// TIA Portal V17 export
// export: Created 2025-05-22T05:59:44.8642244Z, ExportSetting WithDefaults, DisplayName Totally Integrated Automation Portal, DisplayVersion V17 Update 8, DisplayName TIA Portal Openness, DisplayVersion V17 Update 8, DisplayName TIA Portal Version Control Interface, DisplayVersion V17, DisplayName SINAMICS Startdrive Advanced, DisplayVersion V17 SP2, DisplayName SINAMICS Startdrive G110M, G120, G120C, G120D, G120P, G115D, DisplayVersion V17 SP2, DisplayName SINAMICS Startdrive G130, G150, S120, S150, SINAMICS MV, S210, DisplayVersion V17 SP2, DisplayName STEP 7 Professional, DisplayVersion V17 Update 8, DisplayName SINUMERIK ONE STEP 7 Toolbox, DisplayVersion V17 Update 12, DisplayName SINUMERIK ONE PLC Basic Program Plus, DisplayVersion V17 Update 12, DisplayName SINUMERIK 840D sl STEP 7 Toolbox, DisplayVersion V17 Update 12, DisplayName STEP 7 Safety, DisplayVersion V17 Update 6, DisplayName WinCC Advanced, DisplayVersion V17 Update 8
FUNCTION "FC7341_POWDER_PLC_TO_MACHINE_INTERLOCK" : Void   // FC7341, LAD
{ S7_Optimized_Access := 'TRUE' }
VERSION : 0.1
// stored: AutoNumber false, IsIECCheckEnabled false, SetENOAutomatically false, UDAEnableTagReadback false
   VAR_TEMP
      COUNT_FOR_ERROR : Int;
      RET_VAL_1 : Int;
      "DATE" : DTL;
   END_VAR
   VAR CONSTANT
      FC_NUMBER : DInt := 7341;
   END_VAR
   VAR_TEMP   // added for the SCL form of the ladder/FBD networks
      _w1 : Bool;
   END_VAR
BEGIN

REGION Network 1: LIFE BIT
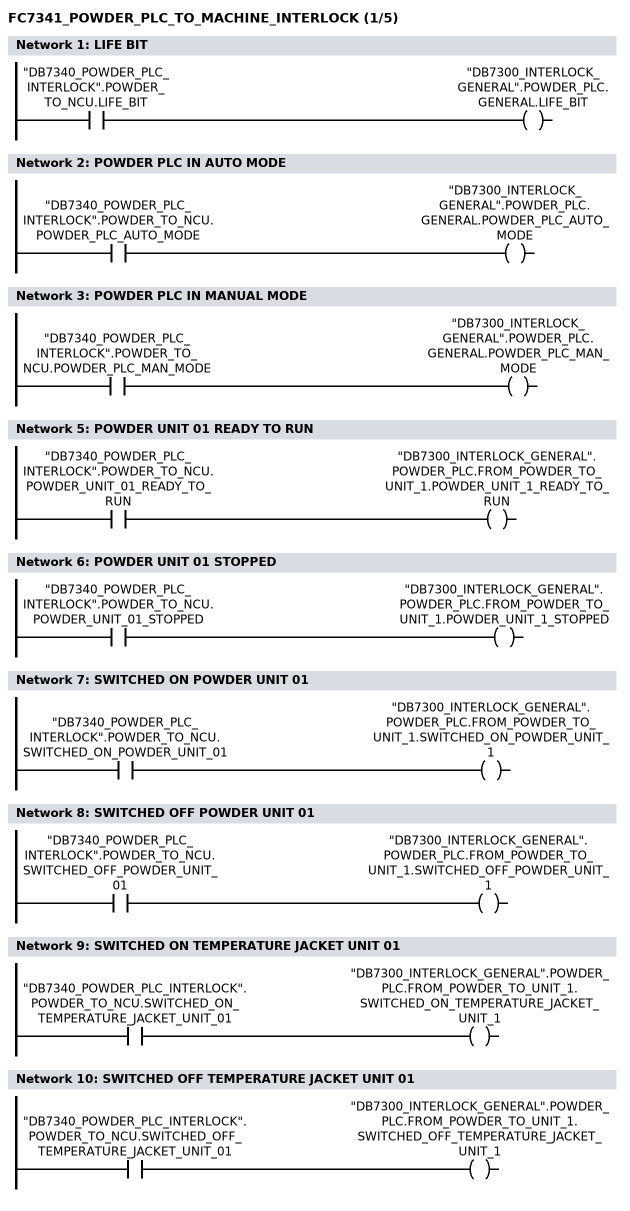
   RUNG wire#powerrail
      Contact( "DB7340_POWDER_PLC_INTERLOCK".POWDER_TO_NCU.LIFE_BIT )
      Coil( "DB7300_INTERLOCK_GENERAL".POWDER_PLC.GENERAL.LIFE_BIT )
   END_RUNG
   // the same network as SCL:
   "DB7300_INTERLOCK_GENERAL".POWDER_PLC.GENERAL.LIFE_BIT := "DB7340_POWDER_PLC_INTERLOCK".POWDER_TO_NCU.LIFE_BIT;
END_REGION

REGION Network 2: POWDER PLC IN AUTO MODE
   RUNG wire#powerrail
      Contact( "DB7340_POWDER_PLC_INTERLOCK".POWDER_TO_NCU.POWDER_PLC_AUTO_MODE )
      Coil( "DB7300_INTERLOCK_GENERAL".POWDER_PLC.GENERAL.POWDER_PLC_AUTO_MODE )
   END_RUNG
   // the same network as SCL:
   "DB7300_INTERLOCK_GENERAL".POWDER_PLC.GENERAL.POWDER_PLC_AUTO_MODE := "DB7340_POWDER_PLC_INTERLOCK".POWDER_TO_NCU.POWDER_PLC_AUTO_MODE;
END_REGION

REGION Network 3: POWDER PLC IN MANUAL MODE
   RUNG wire#powerrail
      Contact( "DB7340_POWDER_PLC_INTERLOCK".POWDER_TO_NCU.POWDER_PLC_MAN_MODE )
      Coil( "DB7300_INTERLOCK_GENERAL".POWDER_PLC.GENERAL.POWDER_PLC_MAN_MODE )
   END_RUNG
   // the same network as SCL:
   "DB7300_INTERLOCK_GENERAL".POWDER_PLC.GENERAL.POWDER_PLC_MAN_MODE := "DB7340_POWDER_PLC_INTERLOCK".POWDER_TO_NCU.POWDER_PLC_MAN_MODE;
END_REGION

REGION Network 4: //////////_UNIT_01_//////////
END_REGION

REGION Network 5: POWDER UNIT 01 READY TO RUN
   RUNG wire#powerrail
      Contact( "DB7340_POWDER_PLC_INTERLOCK".POWDER_TO_NCU.POWDER_UNIT_01_READY_TO_RUN )
      Coil( "DB7300_INTERLOCK_GENERAL".POWDER_PLC.FROM_POWDER_TO_UNIT_1.POWDER_UNIT_1_READY_TO_RUN )
   END_RUNG
   // the same network as SCL:
   "DB7300_INTERLOCK_GENERAL".POWDER_PLC.FROM_POWDER_TO_UNIT_1.POWDER_UNIT_1_READY_TO_RUN := "DB7340_POWDER_PLC_INTERLOCK".POWDER_TO_NCU.POWDER_UNIT_01_READY_TO_RUN;
END_REGION

REGION Network 6: POWDER UNIT 01 STOPPED
   RUNG wire#powerrail
      Contact( "DB7340_POWDER_PLC_INTERLOCK".POWDER_TO_NCU.POWDER_UNIT_01_STOPPED )
      Coil( "DB7300_INTERLOCK_GENERAL".POWDER_PLC.FROM_POWDER_TO_UNIT_1.POWDER_UNIT_1_STOPPED )
   END_RUNG
   // the same network as SCL:
   "DB7300_INTERLOCK_GENERAL".POWDER_PLC.FROM_POWDER_TO_UNIT_1.POWDER_UNIT_1_STOPPED := "DB7340_POWDER_PLC_INTERLOCK".POWDER_TO_NCU.POWDER_UNIT_01_STOPPED;
END_REGION

REGION Network 7: SWITCHED ON POWDER UNIT 01
   RUNG wire#powerrail
      Contact( "DB7340_POWDER_PLC_INTERLOCK".POWDER_TO_NCU.SWITCHED_ON_POWDER_UNIT_01 )
      Coil( "DB7300_INTERLOCK_GENERAL".POWDER_PLC.FROM_POWDER_TO_UNIT_1.SWITCHED_ON_POWDER_UNIT_1 )
   END_RUNG
   // the same network as SCL:
   "DB7300_INTERLOCK_GENERAL".POWDER_PLC.FROM_POWDER_TO_UNIT_1.SWITCHED_ON_POWDER_UNIT_1 := "DB7340_POWDER_PLC_INTERLOCK".POWDER_TO_NCU.SWITCHED_ON_POWDER_UNIT_01;
END_REGION

REGION Network 8: SWITCHED OFF POWDER UNIT 01
   RUNG wire#powerrail
      Contact( "DB7340_POWDER_PLC_INTERLOCK".POWDER_TO_NCU.SWITCHED_OFF_POWDER_UNIT_01 )
      Coil( "DB7300_INTERLOCK_GENERAL".POWDER_PLC.FROM_POWDER_TO_UNIT_1.SWITCHED_OFF_POWDER_UNIT_1 )
   END_RUNG
   // the same network as SCL:
   "DB7300_INTERLOCK_GENERAL".POWDER_PLC.FROM_POWDER_TO_UNIT_1.SWITCHED_OFF_POWDER_UNIT_1 := "DB7340_POWDER_PLC_INTERLOCK".POWDER_TO_NCU.SWITCHED_OFF_POWDER_UNIT_01;
END_REGION

REGION Network 9: SWITCHED ON TEMPERATURE JACKET UNIT 01
   RUNG wire#powerrail
      Contact( "DB7340_POWDER_PLC_INTERLOCK".POWDER_TO_NCU.SWITCHED_ON_TEMPERATURE_JACKET_UNIT_01 )
      Coil( "DB7300_INTERLOCK_GENERAL".POWDER_PLC.FROM_POWDER_TO_UNIT_1.SWITCHED_ON_TEMPERATURE_JACKET_UNIT_1 )
   END_RUNG
   // the same network as SCL:
   "DB7300_INTERLOCK_GENERAL".POWDER_PLC.FROM_POWDER_TO_UNIT_1.SWITCHED_ON_TEMPERATURE_JACKET_UNIT_1 := "DB7340_POWDER_PLC_INTERLOCK".POWDER_TO_NCU.SWITCHED_ON_TEMPERATURE_JACKET_UNIT_01;
END_REGION

REGION Network 10: SWITCHED OFF TEMPERATURE JACKET UNIT 01
   RUNG wire#powerrail
      Contact( "DB7340_POWDER_PLC_INTERLOCK".POWDER_TO_NCU.SWITCHED_OFF_TEMPERATURE_JACKET_UNIT_01 )
      Coil( "DB7300_INTERLOCK_GENERAL".POWDER_PLC.FROM_POWDER_TO_UNIT_1.SWITCHED_OFF_TEMPERATURE_JACKET_UNIT_1 )
   END_RUNG
   // the same network as SCL:
   "DB7300_INTERLOCK_GENERAL".POWDER_PLC.FROM_POWDER_TO_UNIT_1.SWITCHED_OFF_TEMPERATURE_JACKET_UNIT_1 := "DB7340_POWDER_PLC_INTERLOCK".POWDER_TO_NCU.SWITCHED_OFF_TEMPERATURE_JACKET_UNIT_01;
END_REGION

REGION Network 11: UNIT 1 POWDER FEEDER 1 LINE 1 LOW POWDER LEVEL
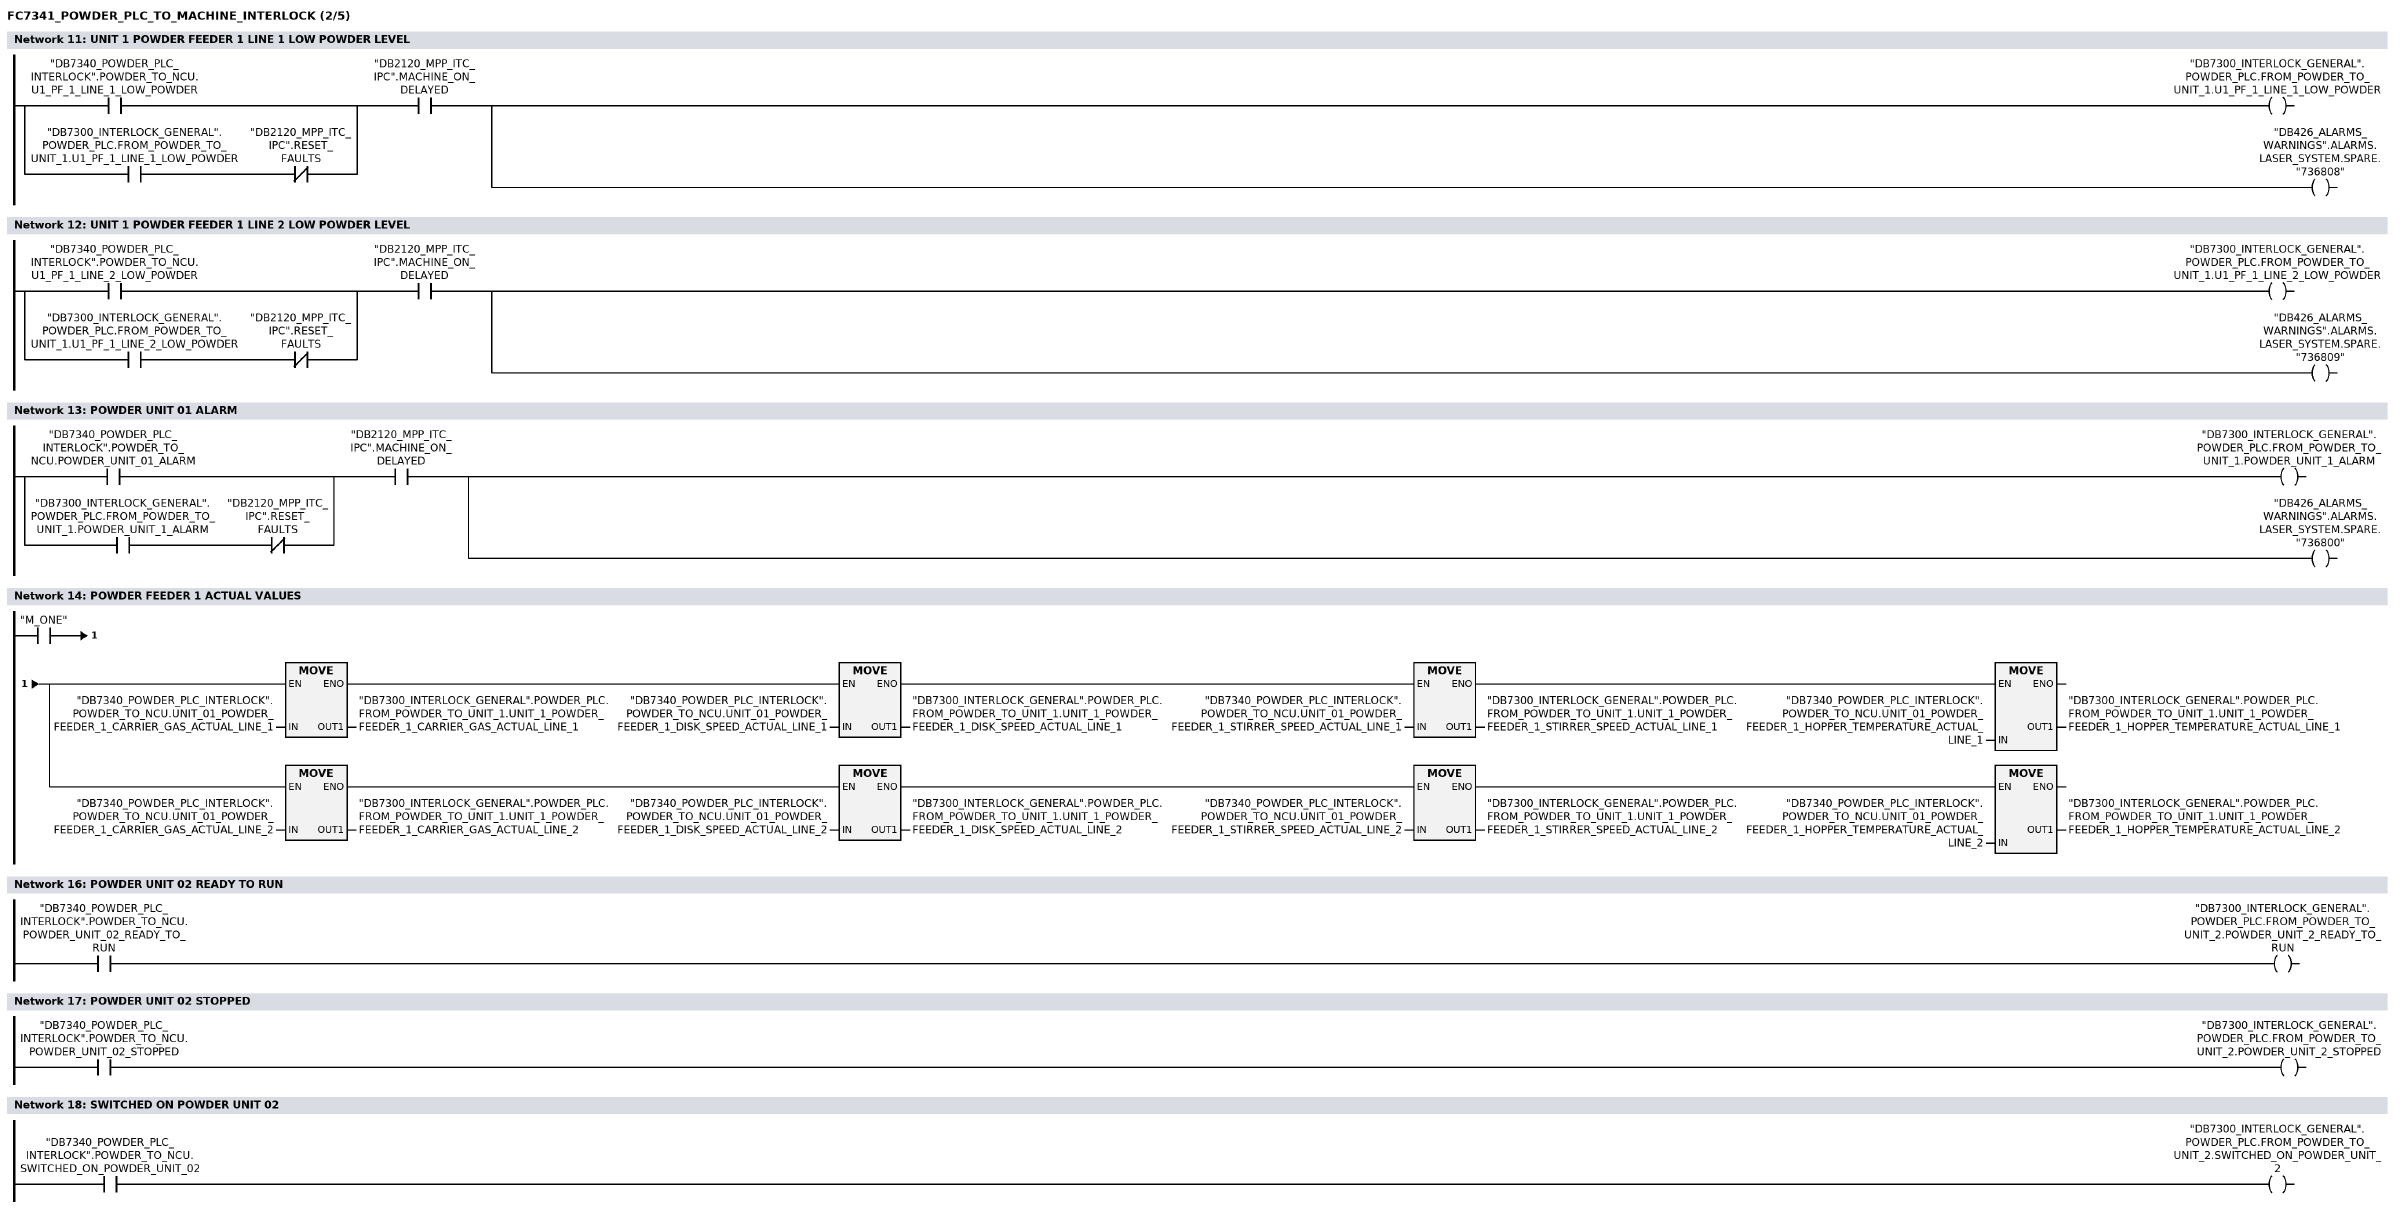
   RUNG wire#powerrail
      Contact( "DB7340_POWDER_PLC_INTERLOCK".POWDER_TO_NCU.U1_PF_1_LINE_1_LOW_POWDER )
      wire#w1
      Contact( "DB2120_MPP_ITC_IPC".MACHINE_ON_DELAYED )
      wire#w2
      Coil( "DB7300_INTERLOCK_GENERAL".POWDER_PLC.FROM_POWDER_TO_UNIT_1.U1_PF_1_LINE_1_LOW_POWDER )
   END_RUNG
   RUNG wire#powerrail
      Contact( "DB7300_INTERLOCK_GENERAL".POWDER_PLC.FROM_POWDER_TO_UNIT_1.U1_PF_1_LINE_1_LOW_POWDER )
      I_Contact( "DB2120_MPP_ITC_IPC".RESET_FAULTS )
   END_RUNG wire#w1
   RUNG wire#w2
      Coil( "DB426_ALARMS_WARNINGS".ALARMS.LASER_SYSTEM.SPARE."736808" )
   END_RUNG
   // the same network as SCL:
   "DB7300_INTERLOCK_GENERAL".POWDER_PLC.FROM_POWDER_TO_UNIT_1.U1_PF_1_LINE_1_LOW_POWDER := ("DB7340_POWDER_PLC_INTERLOCK".POWDER_TO_NCU.U1_PF_1_LINE_1_LOW_POWDER OR ("DB7300_INTERLOCK_GENERAL".POWDER_PLC.FROM_POWDER_TO_UNIT_1.U1_PF_1_LINE_1_LOW_POWDER AND NOT "DB2120_MPP_ITC_IPC".RESET_FAULTS)) AND "DB2120_MPP_ITC_IPC".MACHINE_ON_DELAYED;
   "DB426_ALARMS_WARNINGS".ALARMS.LASER_SYSTEM.SPARE."736808" := "DB7300_INTERLOCK_GENERAL".POWDER_PLC.FROM_POWDER_TO_UNIT_1.U1_PF_1_LINE_1_LOW_POWDER;
END_REGION

REGION Network 12: UNIT 1 POWDER FEEDER 1 LINE 2 LOW POWDER LEVEL
   RUNG wire#powerrail
      Contact( "DB7340_POWDER_PLC_INTERLOCK".POWDER_TO_NCU.U1_PF_1_LINE_2_LOW_POWDER )
      wire#w1
      Contact( "DB2120_MPP_ITC_IPC".MACHINE_ON_DELAYED )
      wire#w2
      Coil( "DB7300_INTERLOCK_GENERAL".POWDER_PLC.FROM_POWDER_TO_UNIT_1.U1_PF_1_LINE_2_LOW_POWDER )
   END_RUNG
   RUNG wire#powerrail
      Contact( "DB7300_INTERLOCK_GENERAL".POWDER_PLC.FROM_POWDER_TO_UNIT_1.U1_PF_1_LINE_2_LOW_POWDER )
      I_Contact( "DB2120_MPP_ITC_IPC".RESET_FAULTS )
   END_RUNG wire#w1
   RUNG wire#w2
      Coil( "DB426_ALARMS_WARNINGS".ALARMS.LASER_SYSTEM.SPARE."736809" )
   END_RUNG
   // the same network as SCL:
   "DB7300_INTERLOCK_GENERAL".POWDER_PLC.FROM_POWDER_TO_UNIT_1.U1_PF_1_LINE_2_LOW_POWDER := ("DB7340_POWDER_PLC_INTERLOCK".POWDER_TO_NCU.U1_PF_1_LINE_2_LOW_POWDER OR ("DB7300_INTERLOCK_GENERAL".POWDER_PLC.FROM_POWDER_TO_UNIT_1.U1_PF_1_LINE_2_LOW_POWDER AND NOT "DB2120_MPP_ITC_IPC".RESET_FAULTS)) AND "DB2120_MPP_ITC_IPC".MACHINE_ON_DELAYED;
   "DB426_ALARMS_WARNINGS".ALARMS.LASER_SYSTEM.SPARE."736809" := "DB7300_INTERLOCK_GENERAL".POWDER_PLC.FROM_POWDER_TO_UNIT_1.U1_PF_1_LINE_2_LOW_POWDER;
END_REGION

REGION Network 13: POWDER UNIT 01 ALARM
   RUNG wire#powerrail
      Contact( "DB7340_POWDER_PLC_INTERLOCK".POWDER_TO_NCU.POWDER_UNIT_01_ALARM )
      wire#w1
      Contact( "DB2120_MPP_ITC_IPC".MACHINE_ON_DELAYED )
      wire#w2
      Coil( "DB7300_INTERLOCK_GENERAL".POWDER_PLC.FROM_POWDER_TO_UNIT_1.POWDER_UNIT_1_ALARM )
   END_RUNG
   RUNG wire#powerrail
      Contact( "DB7300_INTERLOCK_GENERAL".POWDER_PLC.FROM_POWDER_TO_UNIT_1.POWDER_UNIT_1_ALARM )
      I_Contact( "DB2120_MPP_ITC_IPC".RESET_FAULTS )
   END_RUNG wire#w1
   RUNG wire#w2
      Coil( "DB426_ALARMS_WARNINGS".ALARMS.LASER_SYSTEM.SPARE."736800" )
   END_RUNG
   // the same network as SCL:
   "DB7300_INTERLOCK_GENERAL".POWDER_PLC.FROM_POWDER_TO_UNIT_1.POWDER_UNIT_1_ALARM := ("DB7340_POWDER_PLC_INTERLOCK".POWDER_TO_NCU.POWDER_UNIT_01_ALARM OR ("DB7300_INTERLOCK_GENERAL".POWDER_PLC.FROM_POWDER_TO_UNIT_1.POWDER_UNIT_1_ALARM AND NOT "DB2120_MPP_ITC_IPC".RESET_FAULTS)) AND "DB2120_MPP_ITC_IPC".MACHINE_ON_DELAYED;
   "DB426_ALARMS_WARNINGS".ALARMS.LASER_SYSTEM.SPARE."736800" := "DB7300_INTERLOCK_GENERAL".POWDER_PLC.FROM_POWDER_TO_UNIT_1.POWDER_UNIT_1_ALARM;
END_REGION

REGION Network 14: POWDER FEEDER 1 ACTUAL VALUES
   RUNG wire#powerrail
      Contact( "M_ONE" )
      wire#w1
      Move(in := "DB7340_POWDER_PLC_INTERLOCK".POWDER_TO_NCU.UNIT_01_POWDER_FEEDER_1_CARRIER_GAS_ACTUAL_LINE_1, out1 => "DB7300_INTERLOCK_GENERAL".POWDER_PLC.FROM_POWDER_TO_UNIT_1.UNIT_1_POWDER_FEEDER_1_CARRIER_GAS_ACTUAL_LINE_1)
      Move(in := "DB7340_POWDER_PLC_INTERLOCK".POWDER_TO_NCU.UNIT_01_POWDER_FEEDER_1_DISK_SPEED_ACTUAL_LINE_1, out1 => "DB7300_INTERLOCK_GENERAL".POWDER_PLC.FROM_POWDER_TO_UNIT_1.UNIT_1_POWDER_FEEDER_1_DISK_SPEED_ACTUAL_LINE_1)
      Move(in := "DB7340_POWDER_PLC_INTERLOCK".POWDER_TO_NCU.UNIT_01_POWDER_FEEDER_1_STIRRER_SPEED_ACTUAL_LINE_1, out1 => "DB7300_INTERLOCK_GENERAL".POWDER_PLC.FROM_POWDER_TO_UNIT_1.UNIT_1_POWDER_FEEDER_1_STIRRER_SPEED_ACTUAL_LINE_1)
      Move(in := "DB7340_POWDER_PLC_INTERLOCK".POWDER_TO_NCU.UNIT_01_POWDER_FEEDER_1_HOPPER_TEMPERATURE_ACTUAL_LINE_1, out1 => "DB7300_INTERLOCK_GENERAL".POWDER_PLC.FROM_POWDER_TO_UNIT_1.UNIT_1_POWDER_FEEDER_1_HOPPER_TEMPERATURE_ACTUAL_LINE_1)
   END_RUNG
   RUNG wire#w1
      Move(in := "DB7340_POWDER_PLC_INTERLOCK".POWDER_TO_NCU.UNIT_01_POWDER_FEEDER_1_CARRIER_GAS_ACTUAL_LINE_2, out1 => "DB7300_INTERLOCK_GENERAL".POWDER_PLC.FROM_POWDER_TO_UNIT_1.UNIT_1_POWDER_FEEDER_1_CARRIER_GAS_ACTUAL_LINE_2)
      Move(in := "DB7340_POWDER_PLC_INTERLOCK".POWDER_TO_NCU.UNIT_01_POWDER_FEEDER_1_DISK_SPEED_ACTUAL_LINE_2, out1 => "DB7300_INTERLOCK_GENERAL".POWDER_PLC.FROM_POWDER_TO_UNIT_1.UNIT_1_POWDER_FEEDER_1_DISK_SPEED_ACTUAL_LINE_2)
      Move(in := "DB7340_POWDER_PLC_INTERLOCK".POWDER_TO_NCU.UNIT_01_POWDER_FEEDER_1_STIRRER_SPEED_ACTUAL_LINE_2, out1 => "DB7300_INTERLOCK_GENERAL".POWDER_PLC.FROM_POWDER_TO_UNIT_1.UNIT_1_POWDER_FEEDER_1_STIRRER_SPEED_ACTUAL_LINE_2)
      Move(in := "DB7340_POWDER_PLC_INTERLOCK".POWDER_TO_NCU.UNIT_01_POWDER_FEEDER_1_HOPPER_TEMPERATURE_ACTUAL_LINE_2, out1 => "DB7300_INTERLOCK_GENERAL".POWDER_PLC.FROM_POWDER_TO_UNIT_1.UNIT_1_POWDER_FEEDER_1_HOPPER_TEMPERATURE_ACTUAL_LINE_2)
   END_RUNG
   // the same network as SCL:
   IF "M_ONE" THEN
       "DB7300_INTERLOCK_GENERAL".POWDER_PLC.FROM_POWDER_TO_UNIT_1.UNIT_1_POWDER_FEEDER_1_CARRIER_GAS_ACTUAL_LINE_1 := "DB7340_POWDER_PLC_INTERLOCK".POWDER_TO_NCU.UNIT_01_POWDER_FEEDER_1_CARRIER_GAS_ACTUAL_LINE_1;
       "DB7300_INTERLOCK_GENERAL".POWDER_PLC.FROM_POWDER_TO_UNIT_1.UNIT_1_POWDER_FEEDER_1_DISK_SPEED_ACTUAL_LINE_1 := "DB7340_POWDER_PLC_INTERLOCK".POWDER_TO_NCU.UNIT_01_POWDER_FEEDER_1_DISK_SPEED_ACTUAL_LINE_1;
       "DB7300_INTERLOCK_GENERAL".POWDER_PLC.FROM_POWDER_TO_UNIT_1.UNIT_1_POWDER_FEEDER_1_STIRRER_SPEED_ACTUAL_LINE_1 := "DB7340_POWDER_PLC_INTERLOCK".POWDER_TO_NCU.UNIT_01_POWDER_FEEDER_1_STIRRER_SPEED_ACTUAL_LINE_1;
       "DB7300_INTERLOCK_GENERAL".POWDER_PLC.FROM_POWDER_TO_UNIT_1.UNIT_1_POWDER_FEEDER_1_HOPPER_TEMPERATURE_ACTUAL_LINE_1 := "DB7340_POWDER_PLC_INTERLOCK".POWDER_TO_NCU.UNIT_01_POWDER_FEEDER_1_HOPPER_TEMPERATURE_ACTUAL_LINE_1;
       "DB7300_INTERLOCK_GENERAL".POWDER_PLC.FROM_POWDER_TO_UNIT_1.UNIT_1_POWDER_FEEDER_1_CARRIER_GAS_ACTUAL_LINE_2 := "DB7340_POWDER_PLC_INTERLOCK".POWDER_TO_NCU.UNIT_01_POWDER_FEEDER_1_CARRIER_GAS_ACTUAL_LINE_2;
       "DB7300_INTERLOCK_GENERAL".POWDER_PLC.FROM_POWDER_TO_UNIT_1.UNIT_1_POWDER_FEEDER_1_DISK_SPEED_ACTUAL_LINE_2 := "DB7340_POWDER_PLC_INTERLOCK".POWDER_TO_NCU.UNIT_01_POWDER_FEEDER_1_DISK_SPEED_ACTUAL_LINE_2;
       "DB7300_INTERLOCK_GENERAL".POWDER_PLC.FROM_POWDER_TO_UNIT_1.UNIT_1_POWDER_FEEDER_1_STIRRER_SPEED_ACTUAL_LINE_2 := "DB7340_POWDER_PLC_INTERLOCK".POWDER_TO_NCU.UNIT_01_POWDER_FEEDER_1_STIRRER_SPEED_ACTUAL_LINE_2;
       "DB7300_INTERLOCK_GENERAL".POWDER_PLC.FROM_POWDER_TO_UNIT_1.UNIT_1_POWDER_FEEDER_1_HOPPER_TEMPERATURE_ACTUAL_LINE_2 := "DB7340_POWDER_PLC_INTERLOCK".POWDER_TO_NCU.UNIT_01_POWDER_FEEDER_1_HOPPER_TEMPERATURE_ACTUAL_LINE_2;
   END_IF;
END_REGION

REGION Network 15: //////////_UNIT_02_//////////
END_REGION

REGION Network 16: POWDER UNIT 02 READY TO RUN
   RUNG wire#powerrail
      Contact( "DB7340_POWDER_PLC_INTERLOCK".POWDER_TO_NCU.POWDER_UNIT_02_READY_TO_RUN )
      Coil( "DB7300_INTERLOCK_GENERAL".POWDER_PLC.FROM_POWDER_TO_UNIT_2.POWDER_UNIT_2_READY_TO_RUN )
   END_RUNG
   // the same network as SCL:
   "DB7300_INTERLOCK_GENERAL".POWDER_PLC.FROM_POWDER_TO_UNIT_2.POWDER_UNIT_2_READY_TO_RUN := "DB7340_POWDER_PLC_INTERLOCK".POWDER_TO_NCU.POWDER_UNIT_02_READY_TO_RUN;
END_REGION

REGION Network 17: POWDER UNIT 02 STOPPED
   RUNG wire#powerrail
      Contact( "DB7340_POWDER_PLC_INTERLOCK".POWDER_TO_NCU.POWDER_UNIT_02_STOPPED )
      Coil( "DB7300_INTERLOCK_GENERAL".POWDER_PLC.FROM_POWDER_TO_UNIT_2.POWDER_UNIT_2_STOPPED )
   END_RUNG
   // the same network as SCL:
   "DB7300_INTERLOCK_GENERAL".POWDER_PLC.FROM_POWDER_TO_UNIT_2.POWDER_UNIT_2_STOPPED := "DB7340_POWDER_PLC_INTERLOCK".POWDER_TO_NCU.POWDER_UNIT_02_STOPPED;
END_REGION

REGION Network 18: SWITCHED ON POWDER UNIT 02
   RUNG wire#powerrail
      Contact( "DB7340_POWDER_PLC_INTERLOCK".POWDER_TO_NCU.SWITCHED_ON_POWDER_UNIT_02 )
      Coil( "DB7300_INTERLOCK_GENERAL".POWDER_PLC.FROM_POWDER_TO_UNIT_2.SWITCHED_ON_POWDER_UNIT_2 )
   END_RUNG
   // the same network as SCL:
   "DB7300_INTERLOCK_GENERAL".POWDER_PLC.FROM_POWDER_TO_UNIT_2.SWITCHED_ON_POWDER_UNIT_2 := "DB7340_POWDER_PLC_INTERLOCK".POWDER_TO_NCU.SWITCHED_ON_POWDER_UNIT_02;
END_REGION

REGION Network 19: SWITCHED OFF POWDER UNIT 02
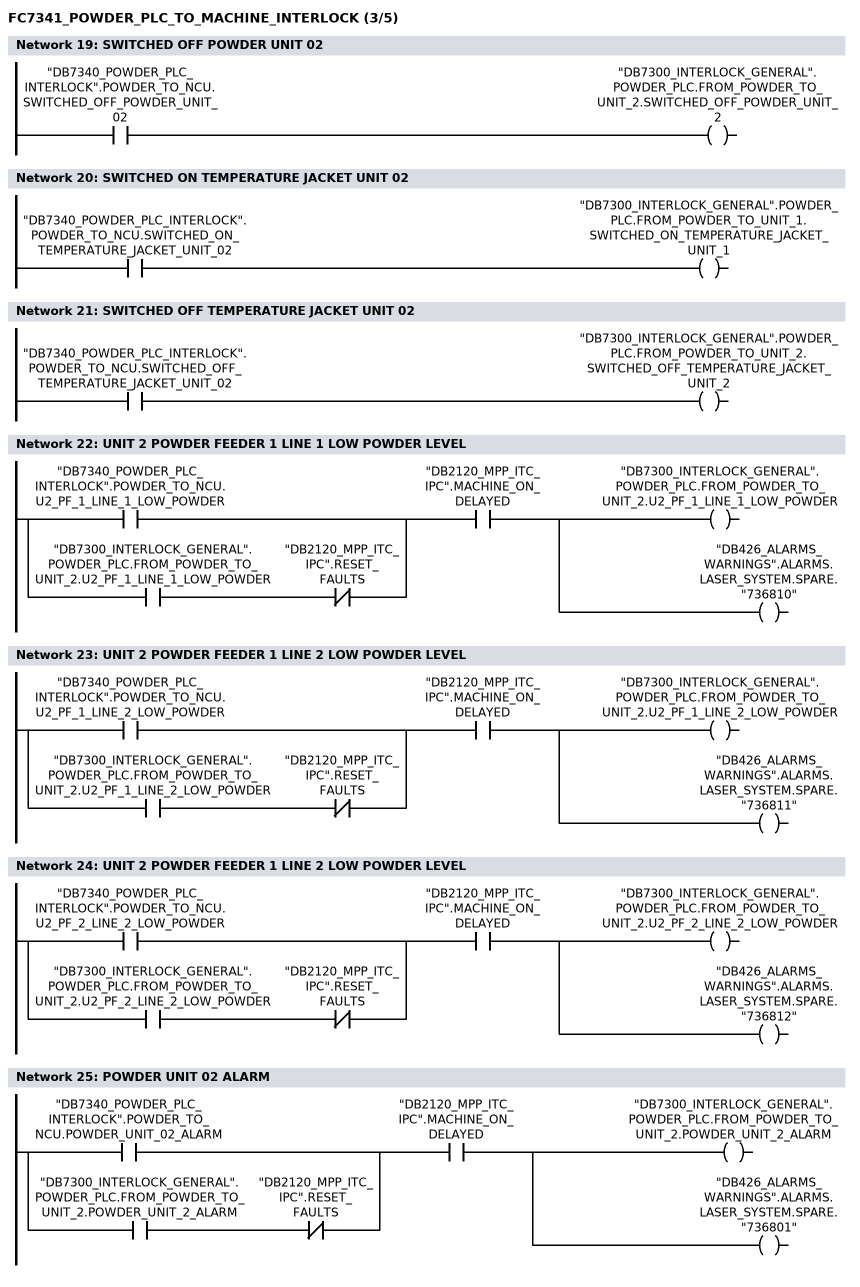
   RUNG wire#powerrail
      Contact( "DB7340_POWDER_PLC_INTERLOCK".POWDER_TO_NCU.SWITCHED_OFF_POWDER_UNIT_02 )
      Coil( "DB7300_INTERLOCK_GENERAL".POWDER_PLC.FROM_POWDER_TO_UNIT_2.SWITCHED_OFF_POWDER_UNIT_2 )
   END_RUNG
   // the same network as SCL:
   "DB7300_INTERLOCK_GENERAL".POWDER_PLC.FROM_POWDER_TO_UNIT_2.SWITCHED_OFF_POWDER_UNIT_2 := "DB7340_POWDER_PLC_INTERLOCK".POWDER_TO_NCU.SWITCHED_OFF_POWDER_UNIT_02;
END_REGION

REGION Network 20: SWITCHED ON TEMPERATURE JACKET UNIT 02
   RUNG wire#powerrail
      Contact( "DB7340_POWDER_PLC_INTERLOCK".POWDER_TO_NCU.SWITCHED_ON_TEMPERATURE_JACKET_UNIT_02 )
      Coil( "DB7300_INTERLOCK_GENERAL".POWDER_PLC.FROM_POWDER_TO_UNIT_1.SWITCHED_ON_TEMPERATURE_JACKET_UNIT_1 )
   END_RUNG
   // the same network as SCL:
   "DB7300_INTERLOCK_GENERAL".POWDER_PLC.FROM_POWDER_TO_UNIT_1.SWITCHED_ON_TEMPERATURE_JACKET_UNIT_1 := "DB7340_POWDER_PLC_INTERLOCK".POWDER_TO_NCU.SWITCHED_ON_TEMPERATURE_JACKET_UNIT_02;
END_REGION

REGION Network 21: SWITCHED OFF TEMPERATURE JACKET UNIT 02
   RUNG wire#powerrail
      Contact( "DB7340_POWDER_PLC_INTERLOCK".POWDER_TO_NCU.SWITCHED_OFF_TEMPERATURE_JACKET_UNIT_02 )
      Coil( "DB7300_INTERLOCK_GENERAL".POWDER_PLC.FROM_POWDER_TO_UNIT_2.SWITCHED_OFF_TEMPERATURE_JACKET_UNIT_2 )
   END_RUNG
   // the same network as SCL:
   "DB7300_INTERLOCK_GENERAL".POWDER_PLC.FROM_POWDER_TO_UNIT_2.SWITCHED_OFF_TEMPERATURE_JACKET_UNIT_2 := "DB7340_POWDER_PLC_INTERLOCK".POWDER_TO_NCU.SWITCHED_OFF_TEMPERATURE_JACKET_UNIT_02;
END_REGION

REGION Network 22: UNIT 2 POWDER FEEDER 1 LINE 1 LOW POWDER LEVEL
   RUNG wire#powerrail
      Contact( "DB7340_POWDER_PLC_INTERLOCK".POWDER_TO_NCU.U2_PF_1_LINE_1_LOW_POWDER )
      wire#w1
      Contact( "DB2120_MPP_ITC_IPC".MACHINE_ON_DELAYED )
      wire#w2
      Coil( "DB7300_INTERLOCK_GENERAL".POWDER_PLC.FROM_POWDER_TO_UNIT_2.U2_PF_1_LINE_1_LOW_POWDER )
   END_RUNG
   RUNG wire#powerrail
      Contact( "DB7300_INTERLOCK_GENERAL".POWDER_PLC.FROM_POWDER_TO_UNIT_2.U2_PF_1_LINE_1_LOW_POWDER )
      I_Contact( "DB2120_MPP_ITC_IPC".RESET_FAULTS )
   END_RUNG wire#w1
   RUNG wire#w2
      Coil( "DB426_ALARMS_WARNINGS".ALARMS.LASER_SYSTEM.SPARE."736810" )
   END_RUNG
   // the same network as SCL:
   "DB7300_INTERLOCK_GENERAL".POWDER_PLC.FROM_POWDER_TO_UNIT_2.U2_PF_1_LINE_1_LOW_POWDER := ("DB7340_POWDER_PLC_INTERLOCK".POWDER_TO_NCU.U2_PF_1_LINE_1_LOW_POWDER OR ("DB7300_INTERLOCK_GENERAL".POWDER_PLC.FROM_POWDER_TO_UNIT_2.U2_PF_1_LINE_1_LOW_POWDER AND NOT "DB2120_MPP_ITC_IPC".RESET_FAULTS)) AND "DB2120_MPP_ITC_IPC".MACHINE_ON_DELAYED;
   "DB426_ALARMS_WARNINGS".ALARMS.LASER_SYSTEM.SPARE."736810" := "DB7300_INTERLOCK_GENERAL".POWDER_PLC.FROM_POWDER_TO_UNIT_2.U2_PF_1_LINE_1_LOW_POWDER;
END_REGION

REGION Network 23: UNIT 2 POWDER FEEDER 1 LINE 2 LOW POWDER LEVEL
   RUNG wire#powerrail
      Contact( "DB7340_POWDER_PLC_INTERLOCK".POWDER_TO_NCU.U2_PF_1_LINE_2_LOW_POWDER )
      wire#w1
      Contact( "DB2120_MPP_ITC_IPC".MACHINE_ON_DELAYED )
      wire#w2
      Coil( "DB7300_INTERLOCK_GENERAL".POWDER_PLC.FROM_POWDER_TO_UNIT_2.U2_PF_1_LINE_2_LOW_POWDER )
   END_RUNG
   RUNG wire#powerrail
      Contact( "DB7300_INTERLOCK_GENERAL".POWDER_PLC.FROM_POWDER_TO_UNIT_2.U2_PF_1_LINE_2_LOW_POWDER )
      I_Contact( "DB2120_MPP_ITC_IPC".RESET_FAULTS )
   END_RUNG wire#w1
   RUNG wire#w2
      Coil( "DB426_ALARMS_WARNINGS".ALARMS.LASER_SYSTEM.SPARE."736811" )
   END_RUNG
   // the same network as SCL:
   "DB7300_INTERLOCK_GENERAL".POWDER_PLC.FROM_POWDER_TO_UNIT_2.U2_PF_1_LINE_2_LOW_POWDER := ("DB7340_POWDER_PLC_INTERLOCK".POWDER_TO_NCU.U2_PF_1_LINE_2_LOW_POWDER OR ("DB7300_INTERLOCK_GENERAL".POWDER_PLC.FROM_POWDER_TO_UNIT_2.U2_PF_1_LINE_2_LOW_POWDER AND NOT "DB2120_MPP_ITC_IPC".RESET_FAULTS)) AND "DB2120_MPP_ITC_IPC".MACHINE_ON_DELAYED;
   "DB426_ALARMS_WARNINGS".ALARMS.LASER_SYSTEM.SPARE."736811" := "DB7300_INTERLOCK_GENERAL".POWDER_PLC.FROM_POWDER_TO_UNIT_2.U2_PF_1_LINE_2_LOW_POWDER;
END_REGION

REGION Network 24: UNIT 2 POWDER FEEDER 1 LINE 2 LOW POWDER LEVEL
   RUNG wire#powerrail
      Contact( "DB7340_POWDER_PLC_INTERLOCK".POWDER_TO_NCU.U2_PF_2_LINE_2_LOW_POWDER )
      wire#w1
      Contact( "DB2120_MPP_ITC_IPC".MACHINE_ON_DELAYED )
      wire#w2
      Coil( "DB7300_INTERLOCK_GENERAL".POWDER_PLC.FROM_POWDER_TO_UNIT_2.U2_PF_2_LINE_2_LOW_POWDER )
   END_RUNG
   RUNG wire#powerrail
      Contact( "DB7300_INTERLOCK_GENERAL".POWDER_PLC.FROM_POWDER_TO_UNIT_2.U2_PF_2_LINE_2_LOW_POWDER )
      I_Contact( "DB2120_MPP_ITC_IPC".RESET_FAULTS )
   END_RUNG wire#w1
   RUNG wire#w2
      Coil( "DB426_ALARMS_WARNINGS".ALARMS.LASER_SYSTEM.SPARE."736812" )
   END_RUNG
   // the same network as SCL:
   "DB7300_INTERLOCK_GENERAL".POWDER_PLC.FROM_POWDER_TO_UNIT_2.U2_PF_2_LINE_2_LOW_POWDER := ("DB7340_POWDER_PLC_INTERLOCK".POWDER_TO_NCU.U2_PF_2_LINE_2_LOW_POWDER OR ("DB7300_INTERLOCK_GENERAL".POWDER_PLC.FROM_POWDER_TO_UNIT_2.U2_PF_2_LINE_2_LOW_POWDER AND NOT "DB2120_MPP_ITC_IPC".RESET_FAULTS)) AND "DB2120_MPP_ITC_IPC".MACHINE_ON_DELAYED;
   "DB426_ALARMS_WARNINGS".ALARMS.LASER_SYSTEM.SPARE."736812" := "DB7300_INTERLOCK_GENERAL".POWDER_PLC.FROM_POWDER_TO_UNIT_2.U2_PF_2_LINE_2_LOW_POWDER;
END_REGION

REGION Network 25: POWDER UNIT 02 ALARM
   RUNG wire#powerrail
      Contact( "DB7340_POWDER_PLC_INTERLOCK".POWDER_TO_NCU.POWDER_UNIT_02_ALARM )
      wire#w1
      Contact( "DB2120_MPP_ITC_IPC".MACHINE_ON_DELAYED )
      wire#w2
      Coil( "DB7300_INTERLOCK_GENERAL".POWDER_PLC.FROM_POWDER_TO_UNIT_2.POWDER_UNIT_2_ALARM )
   END_RUNG
   RUNG wire#powerrail
      Contact( "DB7300_INTERLOCK_GENERAL".POWDER_PLC.FROM_POWDER_TO_UNIT_2.POWDER_UNIT_2_ALARM )
      I_Contact( "DB2120_MPP_ITC_IPC".RESET_FAULTS )
   END_RUNG wire#w1
   RUNG wire#w2
      Coil( "DB426_ALARMS_WARNINGS".ALARMS.LASER_SYSTEM.SPARE."736801" )
   END_RUNG
   // the same network as SCL:
   "DB7300_INTERLOCK_GENERAL".POWDER_PLC.FROM_POWDER_TO_UNIT_2.POWDER_UNIT_2_ALARM := ("DB7340_POWDER_PLC_INTERLOCK".POWDER_TO_NCU.POWDER_UNIT_02_ALARM OR ("DB7300_INTERLOCK_GENERAL".POWDER_PLC.FROM_POWDER_TO_UNIT_2.POWDER_UNIT_2_ALARM AND NOT "DB2120_MPP_ITC_IPC".RESET_FAULTS)) AND "DB2120_MPP_ITC_IPC".MACHINE_ON_DELAYED;
   "DB426_ALARMS_WARNINGS".ALARMS.LASER_SYSTEM.SPARE."736801" := "DB7300_INTERLOCK_GENERAL".POWDER_PLC.FROM_POWDER_TO_UNIT_2.POWDER_UNIT_2_ALARM;
END_REGION

REGION Network 26: POWDER FEEDER 1 ACTUAL VALUES
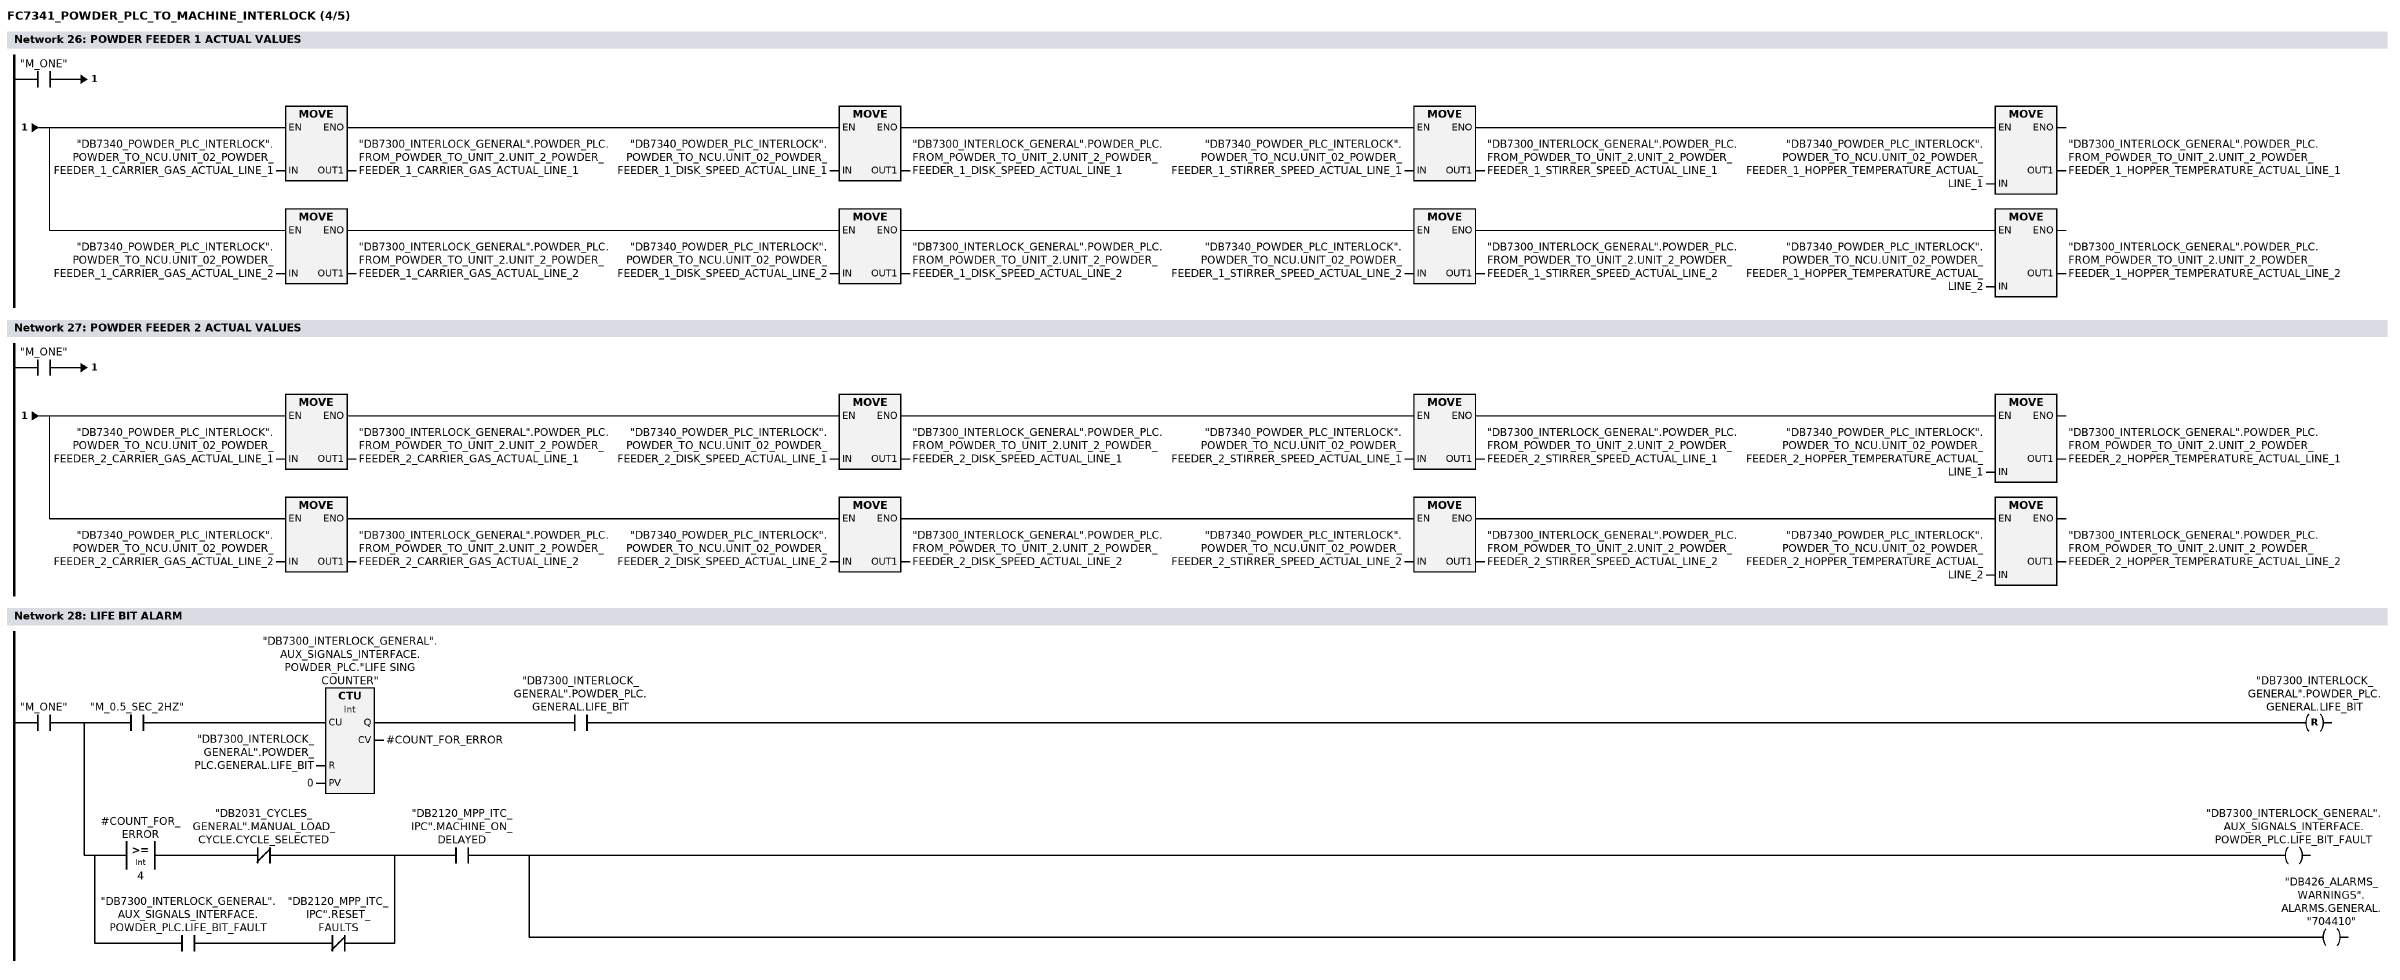
   RUNG wire#powerrail
      Contact( "M_ONE" )
      wire#w1
      Move(in := "DB7340_POWDER_PLC_INTERLOCK".POWDER_TO_NCU.UNIT_02_POWDER_FEEDER_1_CARRIER_GAS_ACTUAL_LINE_1, out1 => "DB7300_INTERLOCK_GENERAL".POWDER_PLC.FROM_POWDER_TO_UNIT_2.UNIT_2_POWDER_FEEDER_1_CARRIER_GAS_ACTUAL_LINE_1)
      Move(in := "DB7340_POWDER_PLC_INTERLOCK".POWDER_TO_NCU.UNIT_02_POWDER_FEEDER_1_DISK_SPEED_ACTUAL_LINE_1, out1 => "DB7300_INTERLOCK_GENERAL".POWDER_PLC.FROM_POWDER_TO_UNIT_2.UNIT_2_POWDER_FEEDER_1_DISK_SPEED_ACTUAL_LINE_1)
      Move(in := "DB7340_POWDER_PLC_INTERLOCK".POWDER_TO_NCU.UNIT_02_POWDER_FEEDER_1_STIRRER_SPEED_ACTUAL_LINE_1, out1 => "DB7300_INTERLOCK_GENERAL".POWDER_PLC.FROM_POWDER_TO_UNIT_2.UNIT_2_POWDER_FEEDER_1_STIRRER_SPEED_ACTUAL_LINE_1)
      Move(in := "DB7340_POWDER_PLC_INTERLOCK".POWDER_TO_NCU.UNIT_02_POWDER_FEEDER_1_HOPPER_TEMPERATURE_ACTUAL_LINE_1, out1 => "DB7300_INTERLOCK_GENERAL".POWDER_PLC.FROM_POWDER_TO_UNIT_2.UNIT_2_POWDER_FEEDER_1_HOPPER_TEMPERATURE_ACTUAL_LINE_1)
   END_RUNG
   RUNG wire#w1
      Move(in := "DB7340_POWDER_PLC_INTERLOCK".POWDER_TO_NCU.UNIT_02_POWDER_FEEDER_1_CARRIER_GAS_ACTUAL_LINE_2, out1 => "DB7300_INTERLOCK_GENERAL".POWDER_PLC.FROM_POWDER_TO_UNIT_2.UNIT_2_POWDER_FEEDER_1_CARRIER_GAS_ACTUAL_LINE_2)
      Move(in := "DB7340_POWDER_PLC_INTERLOCK".POWDER_TO_NCU.UNIT_02_POWDER_FEEDER_1_DISK_SPEED_ACTUAL_LINE_2, out1 => "DB7300_INTERLOCK_GENERAL".POWDER_PLC.FROM_POWDER_TO_UNIT_2.UNIT_2_POWDER_FEEDER_1_DISK_SPEED_ACTUAL_LINE_2)
      Move(in := "DB7340_POWDER_PLC_INTERLOCK".POWDER_TO_NCU.UNIT_02_POWDER_FEEDER_1_STIRRER_SPEED_ACTUAL_LINE_2, out1 => "DB7300_INTERLOCK_GENERAL".POWDER_PLC.FROM_POWDER_TO_UNIT_2.UNIT_2_POWDER_FEEDER_1_STIRRER_SPEED_ACTUAL_LINE_2)
      Move(in := "DB7340_POWDER_PLC_INTERLOCK".POWDER_TO_NCU.UNIT_02_POWDER_FEEDER_1_HOPPER_TEMPERATURE_ACTUAL_LINE_2, out1 => "DB7300_INTERLOCK_GENERAL".POWDER_PLC.FROM_POWDER_TO_UNIT_2.UNIT_2_POWDER_FEEDER_1_HOPPER_TEMPERATURE_ACTUAL_LINE_2)
   END_RUNG
   // the same network as SCL:
   IF "M_ONE" THEN
       "DB7300_INTERLOCK_GENERAL".POWDER_PLC.FROM_POWDER_TO_UNIT_2.UNIT_2_POWDER_FEEDER_1_CARRIER_GAS_ACTUAL_LINE_1 := "DB7340_POWDER_PLC_INTERLOCK".POWDER_TO_NCU.UNIT_02_POWDER_FEEDER_1_CARRIER_GAS_ACTUAL_LINE_1;
       "DB7300_INTERLOCK_GENERAL".POWDER_PLC.FROM_POWDER_TO_UNIT_2.UNIT_2_POWDER_FEEDER_1_DISK_SPEED_ACTUAL_LINE_1 := "DB7340_POWDER_PLC_INTERLOCK".POWDER_TO_NCU.UNIT_02_POWDER_FEEDER_1_DISK_SPEED_ACTUAL_LINE_1;
       "DB7300_INTERLOCK_GENERAL".POWDER_PLC.FROM_POWDER_TO_UNIT_2.UNIT_2_POWDER_FEEDER_1_STIRRER_SPEED_ACTUAL_LINE_1 := "DB7340_POWDER_PLC_INTERLOCK".POWDER_TO_NCU.UNIT_02_POWDER_FEEDER_1_STIRRER_SPEED_ACTUAL_LINE_1;
       "DB7300_INTERLOCK_GENERAL".POWDER_PLC.FROM_POWDER_TO_UNIT_2.UNIT_2_POWDER_FEEDER_1_HOPPER_TEMPERATURE_ACTUAL_LINE_1 := "DB7340_POWDER_PLC_INTERLOCK".POWDER_TO_NCU.UNIT_02_POWDER_FEEDER_1_HOPPER_TEMPERATURE_ACTUAL_LINE_1;
       "DB7300_INTERLOCK_GENERAL".POWDER_PLC.FROM_POWDER_TO_UNIT_2.UNIT_2_POWDER_FEEDER_1_CARRIER_GAS_ACTUAL_LINE_2 := "DB7340_POWDER_PLC_INTERLOCK".POWDER_TO_NCU.UNIT_02_POWDER_FEEDER_1_CARRIER_GAS_ACTUAL_LINE_2;
       "DB7300_INTERLOCK_GENERAL".POWDER_PLC.FROM_POWDER_TO_UNIT_2.UNIT_2_POWDER_FEEDER_1_DISK_SPEED_ACTUAL_LINE_2 := "DB7340_POWDER_PLC_INTERLOCK".POWDER_TO_NCU.UNIT_02_POWDER_FEEDER_1_DISK_SPEED_ACTUAL_LINE_2;
       "DB7300_INTERLOCK_GENERAL".POWDER_PLC.FROM_POWDER_TO_UNIT_2.UNIT_2_POWDER_FEEDER_1_STIRRER_SPEED_ACTUAL_LINE_2 := "DB7340_POWDER_PLC_INTERLOCK".POWDER_TO_NCU.UNIT_02_POWDER_FEEDER_1_STIRRER_SPEED_ACTUAL_LINE_2;
       "DB7300_INTERLOCK_GENERAL".POWDER_PLC.FROM_POWDER_TO_UNIT_2.UNIT_2_POWDER_FEEDER_1_HOPPER_TEMPERATURE_ACTUAL_LINE_2 := "DB7340_POWDER_PLC_INTERLOCK".POWDER_TO_NCU.UNIT_02_POWDER_FEEDER_1_HOPPER_TEMPERATURE_ACTUAL_LINE_2;
   END_IF;
END_REGION

REGION Network 27: POWDER FEEDER 2 ACTUAL VALUES
   RUNG wire#powerrail
      Contact( "M_ONE" )
      wire#w1
      Move(in := "DB7340_POWDER_PLC_INTERLOCK".POWDER_TO_NCU.UNIT_02_POWDER_FEEDER_2_CARRIER_GAS_ACTUAL_LINE_1, out1 => "DB7300_INTERLOCK_GENERAL".POWDER_PLC.FROM_POWDER_TO_UNIT_2.UNIT_2_POWDER_FEEDER_2_CARRIER_GAS_ACTUAL_LINE_1)
      Move(in := "DB7340_POWDER_PLC_INTERLOCK".POWDER_TO_NCU.UNIT_02_POWDER_FEEDER_2_DISK_SPEED_ACTUAL_LINE_1, out1 => "DB7300_INTERLOCK_GENERAL".POWDER_PLC.FROM_POWDER_TO_UNIT_2.UNIT_2_POWDER_FEEDER_2_DISK_SPEED_ACTUAL_LINE_1)
      Move(in := "DB7340_POWDER_PLC_INTERLOCK".POWDER_TO_NCU.UNIT_02_POWDER_FEEDER_2_STIRRER_SPEED_ACTUAL_LINE_1, out1 => "DB7300_INTERLOCK_GENERAL".POWDER_PLC.FROM_POWDER_TO_UNIT_2.UNIT_2_POWDER_FEEDER_2_STIRRER_SPEED_ACTUAL_LINE_1)
      Move(in := "DB7340_POWDER_PLC_INTERLOCK".POWDER_TO_NCU.UNIT_02_POWDER_FEEDER_2_HOPPER_TEMPERATURE_ACTUAL_LINE_1, out1 => "DB7300_INTERLOCK_GENERAL".POWDER_PLC.FROM_POWDER_TO_UNIT_2.UNIT_2_POWDER_FEEDER_2_HOPPER_TEMPERATURE_ACTUAL_LINE_1)
   END_RUNG
   RUNG wire#w1
      Move(in := "DB7340_POWDER_PLC_INTERLOCK".POWDER_TO_NCU.UNIT_02_POWDER_FEEDER_2_CARRIER_GAS_ACTUAL_LINE_2, out1 => "DB7300_INTERLOCK_GENERAL".POWDER_PLC.FROM_POWDER_TO_UNIT_2.UNIT_2_POWDER_FEEDER_2_CARRIER_GAS_ACTUAL_LINE_2)
      Move(in := "DB7340_POWDER_PLC_INTERLOCK".POWDER_TO_NCU.UNIT_02_POWDER_FEEDER_2_DISK_SPEED_ACTUAL_LINE_2, out1 => "DB7300_INTERLOCK_GENERAL".POWDER_PLC.FROM_POWDER_TO_UNIT_2.UNIT_2_POWDER_FEEDER_2_DISK_SPEED_ACTUAL_LINE_2)
      Move(in := "DB7340_POWDER_PLC_INTERLOCK".POWDER_TO_NCU.UNIT_02_POWDER_FEEDER_2_STIRRER_SPEED_ACTUAL_LINE_2, out1 => "DB7300_INTERLOCK_GENERAL".POWDER_PLC.FROM_POWDER_TO_UNIT_2.UNIT_2_POWDER_FEEDER_2_STIRRER_SPEED_ACTUAL_LINE_2)
      Move(in := "DB7340_POWDER_PLC_INTERLOCK".POWDER_TO_NCU.UNIT_02_POWDER_FEEDER_2_HOPPER_TEMPERATURE_ACTUAL_LINE_2, out1 => "DB7300_INTERLOCK_GENERAL".POWDER_PLC.FROM_POWDER_TO_UNIT_2.UNIT_2_POWDER_FEEDER_2_HOPPER_TEMPERATURE_ACTUAL_LINE_2)
   END_RUNG
   // the same network as SCL:
   IF "M_ONE" THEN
       "DB7300_INTERLOCK_GENERAL".POWDER_PLC.FROM_POWDER_TO_UNIT_2.UNIT_2_POWDER_FEEDER_2_CARRIER_GAS_ACTUAL_LINE_1 := "DB7340_POWDER_PLC_INTERLOCK".POWDER_TO_NCU.UNIT_02_POWDER_FEEDER_2_CARRIER_GAS_ACTUAL_LINE_1;
       "DB7300_INTERLOCK_GENERAL".POWDER_PLC.FROM_POWDER_TO_UNIT_2.UNIT_2_POWDER_FEEDER_2_DISK_SPEED_ACTUAL_LINE_1 := "DB7340_POWDER_PLC_INTERLOCK".POWDER_TO_NCU.UNIT_02_POWDER_FEEDER_2_DISK_SPEED_ACTUAL_LINE_1;
       "DB7300_INTERLOCK_GENERAL".POWDER_PLC.FROM_POWDER_TO_UNIT_2.UNIT_2_POWDER_FEEDER_2_STIRRER_SPEED_ACTUAL_LINE_1 := "DB7340_POWDER_PLC_INTERLOCK".POWDER_TO_NCU.UNIT_02_POWDER_FEEDER_2_STIRRER_SPEED_ACTUAL_LINE_1;
       "DB7300_INTERLOCK_GENERAL".POWDER_PLC.FROM_POWDER_TO_UNIT_2.UNIT_2_POWDER_FEEDER_2_HOPPER_TEMPERATURE_ACTUAL_LINE_1 := "DB7340_POWDER_PLC_INTERLOCK".POWDER_TO_NCU.UNIT_02_POWDER_FEEDER_2_HOPPER_TEMPERATURE_ACTUAL_LINE_1;
       "DB7300_INTERLOCK_GENERAL".POWDER_PLC.FROM_POWDER_TO_UNIT_2.UNIT_2_POWDER_FEEDER_2_CARRIER_GAS_ACTUAL_LINE_2 := "DB7340_POWDER_PLC_INTERLOCK".POWDER_TO_NCU.UNIT_02_POWDER_FEEDER_2_CARRIER_GAS_ACTUAL_LINE_2;
       "DB7300_INTERLOCK_GENERAL".POWDER_PLC.FROM_POWDER_TO_UNIT_2.UNIT_2_POWDER_FEEDER_2_DISK_SPEED_ACTUAL_LINE_2 := "DB7340_POWDER_PLC_INTERLOCK".POWDER_TO_NCU.UNIT_02_POWDER_FEEDER_2_DISK_SPEED_ACTUAL_LINE_2;
       "DB7300_INTERLOCK_GENERAL".POWDER_PLC.FROM_POWDER_TO_UNIT_2.UNIT_2_POWDER_FEEDER_2_STIRRER_SPEED_ACTUAL_LINE_2 := "DB7340_POWDER_PLC_INTERLOCK".POWDER_TO_NCU.UNIT_02_POWDER_FEEDER_2_STIRRER_SPEED_ACTUAL_LINE_2;
       "DB7300_INTERLOCK_GENERAL".POWDER_PLC.FROM_POWDER_TO_UNIT_2.UNIT_2_POWDER_FEEDER_2_HOPPER_TEMPERATURE_ACTUAL_LINE_2 := "DB7340_POWDER_PLC_INTERLOCK".POWDER_TO_NCU.UNIT_02_POWDER_FEEDER_2_HOPPER_TEMPERATURE_ACTUAL_LINE_2;
   END_IF;
END_REGION

REGION Network 28: LIFE BIT ALARM
   RUNG wire#powerrail
      Contact( "M_ONE" )
      wire#w1
      Contact( "M_0.5_SEC_2HZ" )
      { S7_Templates := "value_type := Int" } "DB7300_INTERLOCK_GENERAL".AUX_SIGNALS_INTERFACE.POWDER_PLC."LIFE SING COUNTER".CTU(r := "DB7300_INTERLOCK_GENERAL".POWDER_PLC.GENERAL.LIFE_BIT, pv := 0, cv => #COUNT_FOR_ERROR)
      Contact( "DB7300_INTERLOCK_GENERAL".POWDER_PLC.GENERAL.LIFE_BIT )
      R_Coil( "DB7300_INTERLOCK_GENERAL".POWDER_PLC.GENERAL.LIFE_BIT )
   END_RUNG
   RUNG wire#w1
      { S7_Templates := "SrcType := Int" } GE_Contact(in1 := #COUNT_FOR_ERROR, in2 := 4)
      I_Contact( "DB2031_CYCLES_GENERAL".MANUAL_LOAD_CYCLE.CYCLE_SELECTED )
      wire#w2
      Contact( "DB2120_MPP_ITC_IPC".MACHINE_ON_DELAYED )
      wire#w3
      Coil( "DB7300_INTERLOCK_GENERAL".AUX_SIGNALS_INTERFACE.POWDER_PLC.LIFE_BIT_FAULT )
   END_RUNG
   RUNG wire#w1
      Contact( "DB7300_INTERLOCK_GENERAL".AUX_SIGNALS_INTERFACE.POWDER_PLC.LIFE_BIT_FAULT )
      I_Contact( "DB2120_MPP_ITC_IPC".RESET_FAULTS )
   END_RUNG wire#w2
   RUNG wire#w3
      Coil( "DB426_ALARMS_WARNINGS".ALARMS.GENERAL."704410" )
   END_RUNG
   // the same network as SCL:
   "DB7300_INTERLOCK_GENERAL".AUX_SIGNALS_INTERFACE.POWDER_PLC."LIFE SING COUNTER".CTU(CU := "M_ONE" AND "M_0.5_SEC_2HZ",
                           R := "DB7300_INTERLOCK_GENERAL".POWDER_PLC.GENERAL.LIFE_BIT,
                           PV := 0,
                           CV => #COUNT_FOR_ERROR);
   IF "DB7300_INTERLOCK_GENERAL".AUX_SIGNALS_INTERFACE.POWDER_PLC."LIFE SING COUNTER".Q AND "DB7300_INTERLOCK_GENERAL".POWDER_PLC.GENERAL.LIFE_BIT THEN
       "DB7300_INTERLOCK_GENERAL".POWDER_PLC.GENERAL.LIFE_BIT := FALSE;
   END_IF;
   "DB7300_INTERLOCK_GENERAL".AUX_SIGNALS_INTERFACE.POWDER_PLC.LIFE_BIT_FAULT := "M_ONE" AND (((#COUNT_FOR_ERROR >= 4) AND NOT "DB2031_CYCLES_GENERAL".MANUAL_LOAD_CYCLE.CYCLE_SELECTED) OR ("DB7300_INTERLOCK_GENERAL".AUX_SIGNALS_INTERFACE.POWDER_PLC.LIFE_BIT_FAULT AND NOT "DB2120_MPP_ITC_IPC".RESET_FAULTS)) AND "DB2120_MPP_ITC_IPC".MACHINE_ON_DELAYED;
   "DB426_ALARMS_WARNINGS".ALARMS.GENERAL."704410" := "DB7300_INTERLOCK_GENERAL".AUX_SIGNALS_INTERFACE.POWDER_PLC.LIFE_BIT_FAULT;
END_REGION

REGION Network 29: IMMEDIATE STOP ALARMS
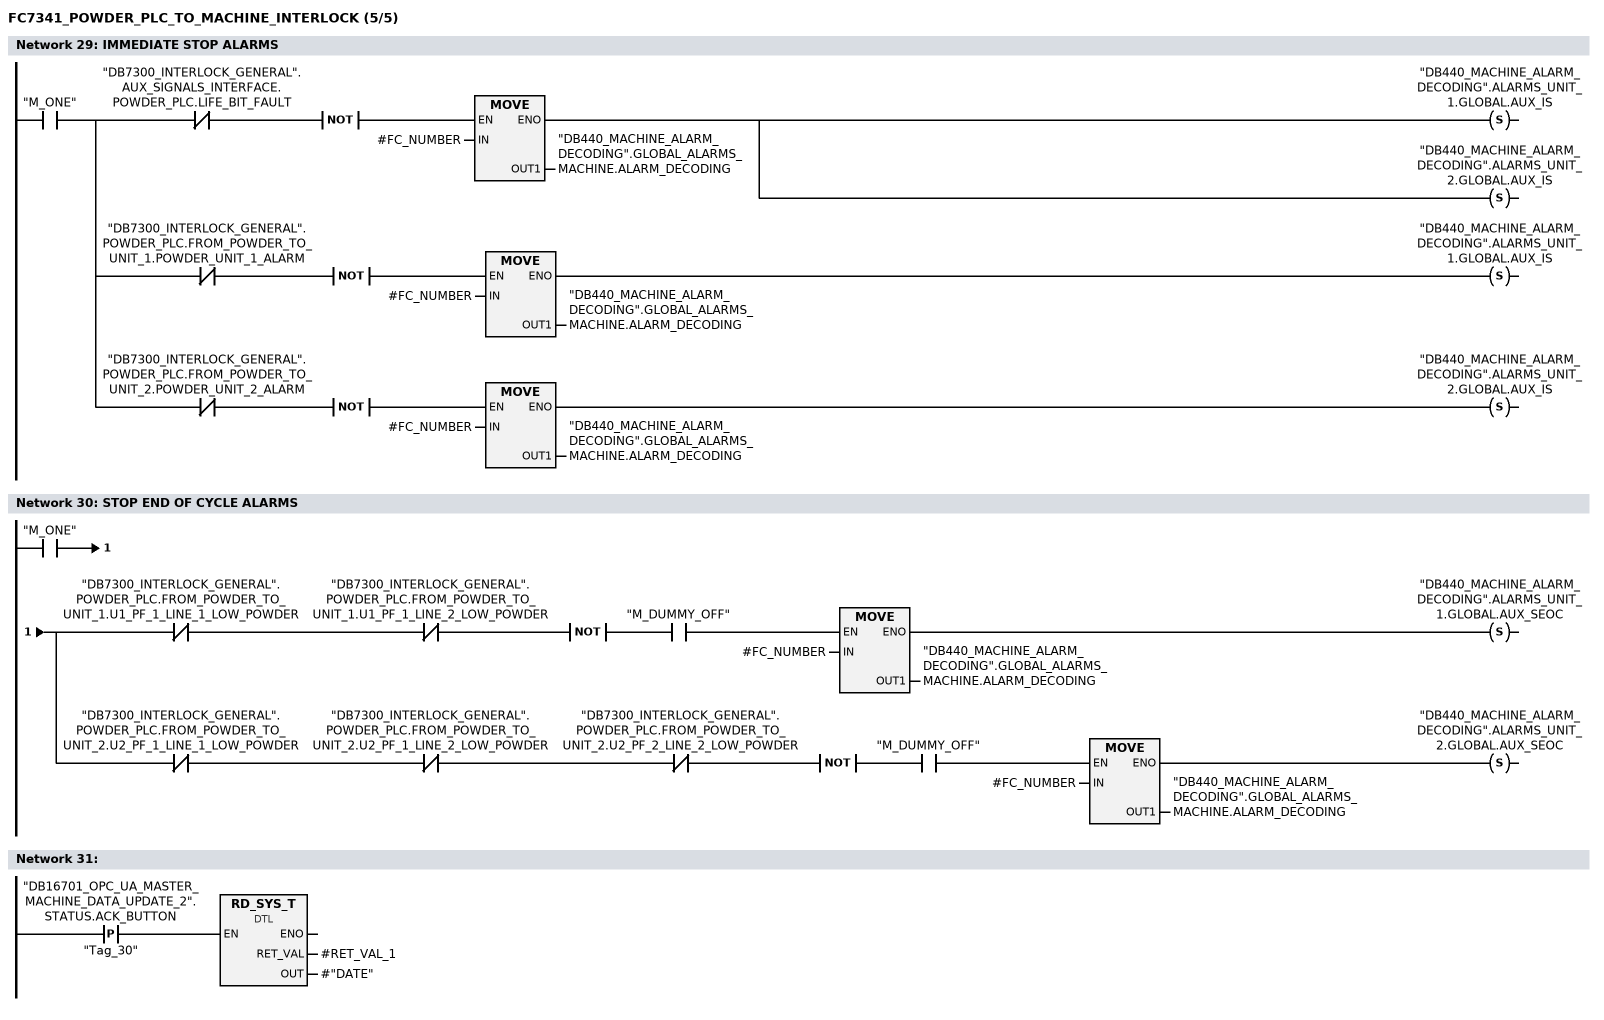
   RUNG wire#powerrail
      Contact( "M_ONE" )
      wire#w1
      I_Contact( "DB7300_INTERLOCK_GENERAL".AUX_SIGNALS_INTERFACE.POWDER_PLC.LIFE_BIT_FAULT )
      Not()
      Move(in := #FC_NUMBER, out1 => "DB440_MACHINE_ALARM_DECODING".GLOBAL_ALARMS_MACHINE.ALARM_DECODING)
      wire#w2
      S_Coil( "DB440_MACHINE_ALARM_DECODING".ALARMS_UNIT_1.GLOBAL.AUX_IS )
   END_RUNG
   RUNG wire#w2
      S_Coil( "DB440_MACHINE_ALARM_DECODING".ALARMS_UNIT_2.GLOBAL.AUX_IS )
   END_RUNG
   RUNG wire#w1
      I_Contact( "DB7300_INTERLOCK_GENERAL".POWDER_PLC.FROM_POWDER_TO_UNIT_1.POWDER_UNIT_1_ALARM )
      Not()
      Move(in := #FC_NUMBER, out1 => "DB440_MACHINE_ALARM_DECODING".GLOBAL_ALARMS_MACHINE.ALARM_DECODING)
      S_Coil( "DB440_MACHINE_ALARM_DECODING".ALARMS_UNIT_1.GLOBAL.AUX_IS )
   END_RUNG
   RUNG wire#w1
      I_Contact( "DB7300_INTERLOCK_GENERAL".POWDER_PLC.FROM_POWDER_TO_UNIT_2.POWDER_UNIT_2_ALARM )
      Not()
      Move(in := #FC_NUMBER, out1 => "DB440_MACHINE_ALARM_DECODING".GLOBAL_ALARMS_MACHINE.ALARM_DECODING)
      S_Coil( "DB440_MACHINE_ALARM_DECODING".ALARMS_UNIT_2.GLOBAL.AUX_IS )
   END_RUNG
   // the same network as SCL:
   IF NOT ("M_ONE" AND NOT "DB7300_INTERLOCK_GENERAL".AUX_SIGNALS_INTERFACE.POWDER_PLC.LIFE_BIT_FAULT) THEN
       "DB440_MACHINE_ALARM_DECODING".GLOBAL_ALARMS_MACHINE.ALARM_DECODING := #FC_NUMBER;
       "DB440_MACHINE_ALARM_DECODING".ALARMS_UNIT_1.GLOBAL.AUX_IS := TRUE;
       "DB440_MACHINE_ALARM_DECODING".ALARMS_UNIT_2.GLOBAL.AUX_IS := TRUE;
   END_IF;
   IF NOT ("M_ONE" AND NOT "DB7300_INTERLOCK_GENERAL".POWDER_PLC.FROM_POWDER_TO_UNIT_1.POWDER_UNIT_1_ALARM) THEN
       "DB440_MACHINE_ALARM_DECODING".GLOBAL_ALARMS_MACHINE.ALARM_DECODING := #FC_NUMBER;
       "DB440_MACHINE_ALARM_DECODING".ALARMS_UNIT_1.GLOBAL.AUX_IS := TRUE;
   END_IF;
   IF NOT ("M_ONE" AND NOT "DB7300_INTERLOCK_GENERAL".POWDER_PLC.FROM_POWDER_TO_UNIT_2.POWDER_UNIT_2_ALARM) THEN
       "DB440_MACHINE_ALARM_DECODING".GLOBAL_ALARMS_MACHINE.ALARM_DECODING := #FC_NUMBER;
       "DB440_MACHINE_ALARM_DECODING".ALARMS_UNIT_2.GLOBAL.AUX_IS := TRUE;
   END_IF;
END_REGION

REGION Network 30: STOP END OF CYCLE ALARMS
   RUNG wire#powerrail
      Contact( "M_ONE" )
      wire#w1
      I_Contact( "DB7300_INTERLOCK_GENERAL".POWDER_PLC.FROM_POWDER_TO_UNIT_1.U1_PF_1_LINE_1_LOW_POWDER )
      I_Contact( "DB7300_INTERLOCK_GENERAL".POWDER_PLC.FROM_POWDER_TO_UNIT_1.U1_PF_1_LINE_2_LOW_POWDER )
      Not()
      Contact( "M_DUMMY_OFF" )
      Move(in := #FC_NUMBER, out1 => "DB440_MACHINE_ALARM_DECODING".GLOBAL_ALARMS_MACHINE.ALARM_DECODING)
      S_Coil( "DB440_MACHINE_ALARM_DECODING".ALARMS_UNIT_1.GLOBAL.AUX_SEOC )
   END_RUNG
   RUNG wire#w1
      I_Contact( "DB7300_INTERLOCK_GENERAL".POWDER_PLC.FROM_POWDER_TO_UNIT_2.U2_PF_1_LINE_1_LOW_POWDER )
      I_Contact( "DB7300_INTERLOCK_GENERAL".POWDER_PLC.FROM_POWDER_TO_UNIT_2.U2_PF_1_LINE_2_LOW_POWDER )
      I_Contact( "DB7300_INTERLOCK_GENERAL".POWDER_PLC.FROM_POWDER_TO_UNIT_2.U2_PF_2_LINE_2_LOW_POWDER )
      Not()
      Contact( "M_DUMMY_OFF" )
      Move(in := #FC_NUMBER, out1 => "DB440_MACHINE_ALARM_DECODING".GLOBAL_ALARMS_MACHINE.ALARM_DECODING)
      S_Coil( "DB440_MACHINE_ALARM_DECODING".ALARMS_UNIT_2.GLOBAL.AUX_SEOC )
   END_RUNG
   // the same network as SCL:
   IF NOT ("M_ONE" AND NOT "DB7300_INTERLOCK_GENERAL".POWDER_PLC.FROM_POWDER_TO_UNIT_1.U1_PF_1_LINE_1_LOW_POWDER AND NOT "DB7300_INTERLOCK_GENERAL".POWDER_PLC.FROM_POWDER_TO_UNIT_1.U1_PF_1_LINE_2_LOW_POWDER) AND "M_DUMMY_OFF" THEN
       "DB440_MACHINE_ALARM_DECODING".GLOBAL_ALARMS_MACHINE.ALARM_DECODING := #FC_NUMBER;
       "DB440_MACHINE_ALARM_DECODING".ALARMS_UNIT_1.GLOBAL.AUX_SEOC := TRUE;
   END_IF;
   IF NOT ("M_ONE" AND NOT "DB7300_INTERLOCK_GENERAL".POWDER_PLC.FROM_POWDER_TO_UNIT_2.U2_PF_1_LINE_1_LOW_POWDER AND NOT "DB7300_INTERLOCK_GENERAL".POWDER_PLC.FROM_POWDER_TO_UNIT_2.U2_PF_1_LINE_2_LOW_POWDER AND NOT "DB7300_INTERLOCK_GENERAL".POWDER_PLC.FROM_POWDER_TO_UNIT_2.U2_PF_2_LINE_2_LOW_POWDER) AND "M_DUMMY_OFF" THEN
       "DB440_MACHINE_ALARM_DECODING".GLOBAL_ALARMS_MACHINE.ALARM_DECODING := #FC_NUMBER;
       "DB440_MACHINE_ALARM_DECODING".ALARMS_UNIT_2.GLOBAL.AUX_SEOC := TRUE;
   END_IF;
END_REGION

REGION Network 31
   RUNG wire#powerrail
      P_Contact(operand := "DB16701_OPC_UA_MASTER_MACHINE_DATA_UPDATE_2".STATUS.ACK_BUTTON, bit := "Tag_30")
      { S7_Templates := "date_type := DTL" } RD_SYS_T(RET_VAL => #RET_VAL_1, OUT => #"DATE")
   END_RUNG
   // the same network as SCL:
   #_w1 := "DB16701_OPC_UA_MASTER_MACHINE_DATA_UPDATE_2".STATUS.ACK_BUTTON AND NOT "Tag_30";   // rising edge of "DB16701_OPC_UA_MASTER_MACHINE_DATA_UPDATE_2".STATUS.ACK_BUTTON
   "Tag_30" := "DB16701_OPC_UA_MASTER_MACHINE_DATA_UPDATE_2".STATUS.ACK_BUTTON;
   IF #_w1 THEN #RET_VAL_1 := RD_SYS_T(OUT => #"DATE"); END_IF;
END_REGION
END_FUNCTION
